(* PLC project Practical Work One, Rexroth ctrlX PLC Engineering ctrlX PLC 1.16.1, author Cedric Lenoir *)
(* stored: creationDateTime 2024-05-03T14:19:29.2185186, version 0.0, modificationDateTime 2024-05-03T14:18:49.029911, organization HEVS *)
(* First Test for Practical Work One *)

TYPE UA_DigitalInput_32 : STRUCT
  Input_0_0 : BOOL;
  Input_0_1 : BOOL;
  Input_0_2 : BOOL;
  Input_0_3 : BOOL;
  Input_0_4 : BOOL;
  Input_0_5 : BOOL;
  Input_0_6 : BOOL;
  Input_0_7 : BOOL;
  Input_1_0 : BOOL;
  Input_1_1 : BOOL;
  Input_1_2 : BOOL;
  Input_1_3 : BOOL;
  Input_1_4 : BOOL;
  Input_1_5 : BOOL;
  Input_1_6 : BOOL;
  Input_1_7 : BOOL;
  Input_2_0 : BOOL;
  Input_2_1 : BOOL;
  Input_2_2 : BOOL;
  Input_2_3 : BOOL;
  Input_2_4 : BOOL;
  Input_2_5 : BOOL;
  Input_2_6 : BOOL;
  Input_2_7 : BOOL;
  Input_3_0 : BOOL;
  Input_3_1 : BOOL;
  Input_3_2 : BOOL;
  Input_3_3 : BOOL;
  Input_3_4 : BOOL;
  Input_3_5 : BOOL;
  Input_3_6 : BOOL;
  Input_3_7 : BOOL;
END_STRUCT;
END_TYPE

TYPE UA_DigitalOutput_32 : STRUCT
  Output_0_0 : BOOL;
  Output_0_1 : BOOL;
  Output_0_2 : BOOL;
  Output_0_3 : BOOL;
  Output_0_4 : BOOL;
  Output_0_5 : BOOL;
  Output_0_6 : BOOL;
  Output_0_7 : BOOL;
  Output_1_0 : BOOL;
  Output_1_1 : BOOL;
  Output_1_2 : BOOL;
  Output_1_3 : BOOL;
  Output_1_4 : BOOL;
  Output_1_5 : BOOL;
  Output_1_6 : BOOL;
  Output_1_7 : BOOL;
  Output_2_0 : BOOL;
  Output_2_1 : BOOL;
  Output_2_2 : BOOL;
  Output_2_3 : BOOL;
  Output_2_4 : BOOL;
  Output_2_5 : BOOL;
  Output_2_6 : BOOL;
  Output_2_7 : BOOL;
  Output_3_0 : BOOL;
  Output_3_1 : BOOL;
  Output_3_2 : BOOL;
  Output_3_3 : BOOL;
  Output_3_4 : BOOL;
  Output_3_5 : BOOL;
  Output_3_6 : BOOL;
  Output_3_7 : BOOL;
END_STRUCT;
END_TYPE

TYPE UA_ButtonAndSignal : STRUCT
  In_Estop : BOOL;
  In_Reset : BOOL;
  In_Start : BOOL;
  In_Stop : BOOL;
  Out_Idle : BOOL;
  Out_Execute : BOOL;
  Out_Stopped : BOOL;
END_STRUCT;
END_TYPE

TYPE UA_O300_DL : STRUCT
  Value : WORD;
  BCD1 : BOOL;
  Q : BOOL;
  A : BOOL;
END_STRUCT;
END_TYPE

TYPE UA_O300_ZL : STRUCT
  BCD1 : BOOL;
  Q : BOOL;
  A : BOOL;
END_STRUCT;
END_TYPE

TYPE UA_U300_D50 : STRUCT
  Value : DWORD;
  Scale : SINT;
  SSC1 : BOOL;
  SSC2 : BOOL;
  Q : BOOL;
  A : BOOL;
  SSC4 : BOOL;
END_STRUCT;
END_TYPE

(* www.hevs.ch Institut Systemes Industriels Project: Projet No: PW Move Absolute Author: Cedric Lenoir Date: 2023 October 16 Summary: List of commands for MoveAbsolute *)
TYPE ST_PlcOpenFbs : STRUCT
  bEnableRemote : BOOL;  (* If TRUE, the FB are driven manually from the HMI *)
  bEnableReadStatus : BOOL;
  bEnableReadPosition : BOOL;
  bEnableReadVelocity : BOOL;
  bMoveAbs : BOOL;
  bStop : BOOL;
  bPowerOn : BOOL;
  bReset : BOOL;
  strGetAxisStatus : STRING;  (* From arAxisStatus_gb[1].Data.PLCopenState; Exist in Data Layer too, s=motion/axs/Axis_X/state/opstate/plcopen *)
END_STRUCT;
END_TYPE

TYPE UA_U300_P50 : STRUCT
  Value : DWORD;
  Scale : SINT;
  SSC1 : BOOL;
  SSC2 : BOOL;
  Q : BOOL;
  A : BOOL;
  SSC4 : BOOL;
END_STRUCT;
END_TYPE

TYPE UA_Schunk_mms : STRUCT
  Value : WORD;
END_STRUCT;
END_TYPE

TYPE UA_Balluf_bcm0002 : STRUCT
  Data_1 : REAL;
  Data_2 : REAL;
  Data_3 : REAL;
  Temperature : REAL;
  Status : DWORD;
END_STRUCT;
END_TYPE

TYPE UA_Festo : STRUCT
  SetOut : BOOL;
END_STRUCT;
END_TYPE

TYPE UA_AnalogIn : STRUCT
  IW_04 : WORD;
  IW_06 : WORD;
  IW_08 : WORD;
  IW_10 : WORD;
  IW_12 : WORD;
  IW_14 : WORD;
  IW_16 : WORD;
  IW_18 : WORD;
END_STRUCT;
END_TYPE

TYPE UA_AnalogOut : STRUCT
  QW_04 : WORD;
  QW_06 : WORD;
  QW_08 : WORD;
  QW_10 : WORD;
END_STRUCT;
END_TYPE

TYPE UA_AboxInterface : STRUCT
  uaButtonAndSignal : UA_ButtonAndSignal;
  uaAnalogIn : UA_AnalogIn;
  uaAnalogOut : UA_AnalogOut;
  uaDigitalIn : UA_DigitalInput_32;
  uaDigitalOut : UA_DigitalOutput_32;
  uaO300_DL_Optic : UA_O300_DL;
  uaO300_ZL_Optic : UA_O300_ZL;
  uaU300_D50_Sound : UA_U300_D50;
  uaU300_P50_Sound : UA_U300_P50;
  uaSchunk : UA_Schunk_mms;
  uaSchunkGripper : UA_Festo;
  uaAccelerometer : UA_Balluf_bcm0002;
END_STRUCT;
END_TYPE

(* www.hevs.ch Institut Systemes Industriels Project: Projet No: PW Move Absolute Author: Cedric Lenoir Date: 2023 October 16 Summary: List of dynamic parameters for Move Absolute *)
TYPE ST_SetMotionParam : STRUCT
  rPosition_mm : LREAL;
  rVeloctiy_mm_s : LREAL;
  rAcceleration_mm_s2 : LREAL;
  rDeceleration_mm_s2 : LREAL;
  rJerk_mm_s3 : LREAL;
END_STRUCT;
END_TYPE

(* www.hevs.ch Institut Systemes Industriels Project: Projet No: PW Move Absolute Author: Cedric Lenoir Date: 2023 October 16 Summary: State Machine Info *)
TYPE ST_StateMachineInfo : STRUCT
  diState : DINT;
  eState : E_Execute;
  strState : STRING;
END_STRUCT;
END_TYPE

{attribute 'qualified_only'}
{attribute 'strict'}
TYPE E_PackStates : (NotActive := 999, Aborted := 10, Clearing := 20, Stopped := 30, Resetting := 40, Idle := 50, Starting := 60, Stopping := 70, Aborting := 80, Execute := 90, Holding := 100, Held := 110, Unholding := 120, Suspending := 200, Suspended := 210, Unsuspending := 220, Completing := 300, Complete := 310) DINT;
END_TYPE

TYPE ST_PackState : STRUCT
  Aborted : BOOL;
  Clearing : BOOL;
  Stopped : BOOL;
  Resetting : BOOL;
  Idle : BOOL;
  Starting : BOOL;
  Stopping : BOOL;
  Aborting : BOOL;
  Execute : BOOL;
  Holding : BOOL;  (* Held Loop *)
  Held : BOOL;
  Unholding : BOOL;
  Suspending : BOOL;  (* Suspended Loop *)
  Suspended : BOOL;
  Unsuspending : BOOL;
  Completing : BOOL;  (* Complete Loop *)
  Complete : BOOL;
END_STRUCT;
END_TYPE

{attribute 'qualified_only'}
{attribute 'strict'}
TYPE E_Clearing : (Idle := 99);
END_TYPE

{attribute 'qualified_only'}
{attribute 'strict'}
TYPE E_Stopping : (Idle := 99);
END_TYPE

{attribute 'qualified_only'}
{attribute 'strict'}
TYPE E_Aborting : (Idle := 99, Disabled := 1, ErrorStop := 2);
END_TYPE

{attribute 'qualified_only'}
{attribute 'strict'}
TYPE E_Resetting : (Idle := 99, eMotionInit := 10, eMotionInitDone := 20);
END_TYPE

{attribute 'qualified_only'}
{attribute 'strict'}
TYPE E_Starting : (Idle := 99, eMotionStarting := 10, eMotionStartingDone := 20, eMotionStartSetPointBack := 22, eMotionStartSetPointBackDone := 23, eMotionSetSynch := 30, eMotionSetSynchDone := 40);
END_TYPE

TYPE ST_RemoteCyclicSetPosition : STRUCT
  in : ST_RemoteCyclicSetPositionIn;  (* Commands for program *)
  out : ST_RemoteCyclicSetPositionOut;  (* Status for program *)
END_STRUCT;
END_TYPE

TYPE ST_RemoteCyclicSetPositionIn : STRUCT
  lrStartPosition_mm : LREAL;  (* Set init position / Start of profile position *)
  lrEndPosition_mm : LREAL;  (* Set end position / End of profile position *)
  udiCycleTimeMultiplier : UDINT := 1000;  (* Cycle Time Multiplier, default is 1000 for 1000 ms *)
  bActivateCoupling : BOOL;  (* Activate coupling, when TRUE, axis position is set by fbGenerateProfile with 5th order polynomial *)
  bStartForward : BOOL;  (* Start polynomial profile forward *)
  bStartBackward : BOOL;  (* Start polynomial profile backward *)
  lrProfileSetPosition : LREAL;  (* Set Position from Profile generator *)
END_STRUCT;
END_TYPE

TYPE ST_RemoteCyclicSetPositionOut : STRUCT
  bInitDone : BOOL;  (* Init done, ready for cyclic motion *)
  bError : BOOL;  (* There is an error *)
  bFwdDone : BOOL;  (* End of cyclic profile Forward *)
  bBackDone : BOOL;  (* End of cyclic profile Back *)
END_STRUCT;
END_TYPE

{attribute 'qualified_only'}
{attribute 'strict'}
TYPE E_Aborted : (Idle := 99, Disabled := 1, ErrorStop := 2);
END_TYPE

(* www.hevs.ch Institut Systemes Industriels Project: Projet No: PW Move Absolute Author: Cedric Lenoir Date: 2024 April 02 Summary: Template of a program using PLCopen on partial Pack State Use a Cyclic Setpoint for motion in Pack Execute. *)
PROGRAM PRG_CyclicSetPoint
  VAR
    uliCount : ULINT;
    bInitDone : BOOL;
    fbPackStates : FB_PackStates;  (* Pack Partial state machine *)
    eAborting : E_Aborting;
    eAborted : E_Aborted;
    eClearing : E_Clearing;
    eResetting : E_Resetting;
    eStarting : E_Starting;
    eStopping : E_Stopping;
    stPlcOpenFbs : ST_PlcOpenFbs;  (* List of Structures *)
    stSetMotionParam : ST_SetMotionParam := (rVeloctiy_mm_s := 2000, rAcceleration_mm_s2 := 1000, rDeceleration_mm_s2 := 1000, rJerk_mm_s3 := 1);
    stStateMachineInfo : ST_StateMachineInfo;
    mcReadActualPosition : MC_ReadActualPosition;  (* List of Function Blocks *)
    mcReadActualVelocity : MC_ReadActualVelocity;
    mcReadStatus : MC_ReadStatus;
    mcPower : MC_Power;
    mcMoveAbsolute : MC_MoveAbsolute;
    mcStop : MC_Stop := (Deceleration := 1);
    mcReset : MC_Reset;
    mcCyclicSetPoint : MB_CyclicSetPoint;
    fbGenerateProfile : FB_GenerateProfile;  (* Set point generator *)
  END_VAR

                    (*
    Some inits independant of the Main State Machine
*)
IF NOT bInitDone THEN
	bInitDone := TRUE;
    stPlcOpenFbs.bEnableReadStatus := TRUE;
    stPlcOpenFbs.bEnableReadPosition := TRUE;
    stPlcOpenFbs.bEnableReadVelocity := TRUE;
END_IF

(*
    Remote conditions
*)
IF stPlcOpenFbs.bEnableRemote THEN
    IF mcMoveAbsolute.Done THEN
        stPlcOpenFbs.bMoveAbs := FALSE;
    END_IF
    IF mcStop.Done THEN
        stPlcOpenFbs.bStop := FALSE;
        stPlcOpenFbs.bMoveAbs := FALSE;
    END_IF
END_IF

// If remote, pack states are disabled
fbPackStates.SoftEstop := mcReadStatus.ErrorStop;
fbPackStates(Enable := NOT stPlcOpenFbs.bEnableRemote,
			 remote := GVL_Abox.uaAboxInterface.uaButtonAndSignal);
			 
(*
	Basically, only Acting state are used, wait state are doing nothing
*)

IF fbPackStates.state.Aborting THEN
	IF mcReadStatus.ErrorStop THEN
		fbPackStates.Aborting_SC := FALSE;
	ELSE
		fbPackStates.Aborting_SC := TRUE;
	END_IF
ELSE
	;
END_IF

IF fbPackStates.state.Aborted THEN
	CASE eAborted OF
		E_Aborted.Idle :
			IF mcReadStatus.Disabled THEN
				eAborted := E_Aborted.Disabled;
			ELSIF mcReadStatus.ErrorStop THEN
				eAborted := E_Aborted.ErrorStop;
			END_IF
		E_Aborted.Disabled :
			IF mcReadStatus.ErrorStop THEN
				eAborted := E_Aborted.ErrorStop;
			END_IF
		E_Aborted.ErrorStop :
			IF mcReadStatus.Disabled THEN
				eAborted := E_Aborted.Disabled;
			END_IF
	END_CASE
ELSE
	eAborted := E_Aborted.Idle;
END_IF

IF fbPackStates.state.Clearing THEN
	IF mcReadStatus.Standstill THEN
		fbPackStates.Clearing_SC := TRUE;
	ELSE
		fbPackStates.Clearing_SC := FALSE;
	END_IF
ELSE
	;
END_IF

IF fbPackStates.state.Stopping THEN
	IF mcReadStatus.Standstill THEN
		fbPackStates.Stopping_SC := TRUE;
	ELSE
		fbPackStates.Stopping_SC := FALSE;
	END_IF
ELSE
	;
END_IF

IF fbPackStates.state.Resetting THEN
	fbPackStates.Resetting_SC := FALSE;
	CASE eResetting OF
		E_Resetting.Idle :
            stSetMotionParam.rPosition_mm := 50;
			stSetMotionParam.rVeloctiy_mm_s := 2000;  
			eResetting := E_Resetting.eMotionInit;

		E_Resetting.eMotionInit :
			IF mcMoveAbsolute.Done THEN
				eResetting := E_Resetting.eMotionInitDone; 
			END_IF

		E_Resetting.eMotionInitDone :
			;;
	END_CASE
	 
	IF eResetting = E_Resetting.eMotionInitDone THEN
		fbPackStates.Resetting_SC := TRUE;
	END_IF
ELSE
	eResetting := E_Resetting.Idle;
END_IF

IF fbPackStates.state.Starting THEN
	fbPackStates.Starting_SC := FALSE;
	CASE eStarting OF
		E_Starting.Idle :
            stSetMotionParam.rPosition_mm := GVL_CyclSetPoint.stRemote.in.lrStartPosition_mm;
			stSetMotionParam.rVeloctiy_mm_s := 2000;  
			eStarting := E_Starting.eMotionStarting;

		E_Starting.eMotionStarting :
			IF mcMoveAbsolute.Done THEN
				eStarting := E_Starting.eMotionStartingDone; 
			END_IF

		E_Starting.eMotionStartingDone :
			IF mcReadStatus.Standstill THEN
				eStarting := E_Starting.eMotionStartSetPointBack;
			END_IF
			
		E_Starting.eMotionStartSetPointBack :
			IF GVL_CyclSetPoint.stRemote.out.bBackDone THEN
				eStarting := E_Starting.eMotionStartSetPointBackDone;
			END_IF
	
		E_Starting.eMotionStartSetPointBackDone :
			eStarting := E_Starting.eMotionSetSynch;

		E_Starting.eMotionSetSynch :
			IF mcReadStatus.DiscreteMotion THEN
				eStarting := E_Starting.eMotionSetSynchDone;
			END_IF
			
		E_Starting.eMotionSetSynchDone :
			;			
			
	END_CASE
	 
	IF eStarting = E_Starting.eMotionSetSynchDone THEN
		fbPackStates.Starting_SC := TRUE;
	END_IF
ELSE
	eStarting := E_Starting.Idle;
END_IF

IF fbPackStates.state.Execute THEN
	fbPackStates.Execute_SC := FALSE;
	(*
		Execute State Machine.
	*)
	CASE stStateMachineInfo.eState OF
		E_Execute.eIdle :
			stStateMachineInfo.strState := 'Idle';
			IF mcCyclicSetPoint.InOperation THEN
				// Set as default value in GVL_CyclSetPoint
				// GVL_CyclSetPoint.stRemote.in.lrEndPosition_mm := 100; 
				stStateMachineInfo.eState := E_Execute.eMotionFwd;
			END_IF

		E_Execute.eMotionFwd :
			stStateMachineInfo.strState := 'Motion One';
			IF GVL_CyclSetPoint.stRemote.out.bFwdDone THEN
				stStateMachineInfo.eState := E_Execute.eMotionFwdDone; 
			END_IF

		E_Execute.eMotionFwdDone :
			stStateMachineInfo.strState := 'Motion One Done';
			IF mcCyclicSetPoint.InOperation THEN
				// Set as default value in GVL_CyclSetPoint
				// GVL_CyclSetPoint.stRemote.in.lrStartPosition_mm := 50;
				stStateMachineInfo.eState := E_Execute.eMotionBack;
			END_IF

		E_Execute.eMotionBack :
			stStateMachineInfo.strState := 'Motion Two';
			IF GVL_CyclSetPoint.stRemote.out.bBackDone THEN
				stStateMachineInfo.eState := E_Execute.eMotionBackDone; 
			END_IF

		E_Execute.eMotionBackDone :
			stStateMachineInfo.strState := 'Motion Two Done'; 
			stStateMachineInfo.eState :=E_Execute.eIdle; 

	END_CASE
	;
ELSE
	stStateMachineInfo.eState := E_Execute.eIdle;
END_IF

IF fbPackStates.state.Holding THEN
	fbPackStates.Holding_SC := TRUE;
ELSE
	;
END_IF

IF fbPackStates.state.Unholding THEN
	fbPackStates.Unholding_SC := TRUE;
ELSE
	;
END_IF

(*
    Get state machine in a DINT format
*)
stStateMachineInfo.diState := stStateMachineInfo.eState;

(*
    Call all Function Blocks at the end of the program
    This is a good practice.
*)
mcReadStatus(Axis := GVL_AxisDefines.X_Axis,
             Enable := stPlcOpenFbs.bEnableReadStatus);

mcReadActualPosition(Axis := GVL_AxisDefines.X_Axis,
                     Enable := stPlcOpenFbs.bEnableReadPosition);
                                         
mcReadActualVelocity(Axis := GVL_AxisDefines.X_Axis,
                     Enable := stPlcOpenFbs.bEnableReadVelocity);

mcPower(Axis := GVL_AxisDefines.X_Axis,
        Enable := (stPlcOpenFbs.bPowerOn AND stPlcOpenFbs.bEnableRemote) OR
                   		NOT stPlcOpenFbs.bEnableRemote AND 
				   		NOT (fbPackStates.state.Aborting OR
                             fbPackStates.state.Aborted));

mcMoveAbsolute(Axis := GVL_AxisDefines.X_Axis,
               Position := stSetMotionParam.rPosition_mm,
               Velocity := stSetMotionParam.rVeloctiy_mm_s,
               Acceleration := stSetMotionParam.rAcceleration_mm_s2,
               Deceleration := stSetMotionParam.rDeceleration_mm_s2,
               Jerk := stSetMotionParam.rJerk_mm_s3,
               Execute := (stPlcOpenFbs.bMoveAbs AND stPlcOpenFbs.bEnableRemote)    OR
                          (eResetting = E_Resetting.eMotionInit)                    OR
						  (eStarting = E_Starting.eMotionStarting));               

// Note that a stop without deceleration leads to an error!!
mcStop(Axis := GVL_AxisDefines.X_Axis,
       Execute := (stPlcOpenFbs.bStop AND stPlcOpenFbs.bEnableRemote) OR
                   fbPackStates.state.Stopping);

mcReset(Axis := GVL_AxisDefines.X_Axis,
        Execute := (stPlcOpenFbs.bReset AND stPlcOpenFbs.bEnableRemote) OR
                    fbPackStates.state.Aborting                         OR
                    eAborted = E_Aborted.ErrorStop);
					
(*
	Set Point Generator
*)
mcCyclicSetPoint.Execute := (stPlcOpenFbs.bEnableRemote AND GVL_CyclSetPoint.stRemote.in.bActivateCoupling) OR
                            (eStarting = E_Starting.eMotionSetSynch);
mcCyclicSetPoint.SetPoint := GVL_CyclSetPoint.stRemote.in.lrProfileSetPosition;
mcCyclicSetPoint(Axis := GVL_AxisDefines.X_Axis);

fbGenerateProfile(bStartForward := (stPlcOpenFbs.bEnableRemote AND GVL_CyclSetPoint.stRemote.in.bStartForward) OR
                                   (stStateMachineInfo.eState = E_Execute.eMotionFwd),
                  bStartBackward := (stPlcOpenFbs.bEnableRemote AND GVL_CyclSetPoint.stRemote.in.bStartBackward) OR
                                    (eStarting = E_Starting.eMotionStartSetPointBack) OR
                                    (stStateMachineInfo.eState = E_Execute.eMotionBack),
                  startPosition_mm := GVL_CyclSetPoint.stRemote.in.lrStartPosition_mm,
                  endPosition_mm := GVL_CyclSetPoint.stRemote.in.lrEndPosition_mm,
                  udiCyclTime_ms := GVL_CyclSetPoint.MOTION_CYCLE_TIME_ms,
                  udiCycleTimeMult := GVL_CyclSetPoint.stRemote.in.udiCycleTimeMultiplier, // Could be a parameter latter when all is working
                  arGoToPos := GVL_CyclSetPoint.arGoToPosition,
                  arReturnFromPos := GVL_CyclSetPoint.arReturnFromPosition,
                  lrSetPosition => GVL_CyclSetPoint.stRemote.in.lrProfileSetPosition,
                  bDoneForward => GVL_CyclSetPoint.stRemote.out.bFwdDone,
                  bDoneBackward => GVL_CyclSetPoint.stRemote.out.bBackDone);					
					
                   
                  
END_PROGRAM

PROGRAM PRG_MapBox
  VAR
    UA_ReadCounterFromStation : DINT;  (* Write from Siemens to ctrX Core Used to check if read is running *)
    UA_ButtonAndSignal_In_Estop : BOOL;
    UA_ButtonAndSignal_In_Reset : BOOL;
    UA_ButtonAndSignal_In_Start : BOOL;
    UA_ButtonAndSignal_In_Stop : BOOL;
    UA_Balluf_bcm0002_Data_1 : REAL;
    UA_Balluf_bcm0002_Data_2 : REAL;
    UA_Balluf_bcm0002_Data_3 : REAL;
    UA_Balluf_bcm0002_Temperature : REAL;
    UA_Balluf_bcm0002_Status : DWORD;
    UA_Festo_SetOut : BOOL;
    UA_O300_DL_Value : WORD;
    UA_O300_DL_BCD1 : BOOL;
    UA_O300_DL_Q : BOOL;
    UA_O300_DL_A : BOOL;
    UA_O300_ZL_BCD1 : BOOL;
    UA_O300_ZL_Q : BOOL;
    UA_O300_ZL_A : BOOL;
    UA_U300_D50_Value : DWORD;
    UA_U300_D50_Scale : SINT;
    UA_U300_D50_SSC1 : BOOL;
    UA_U300_D50_SSC2 : BOOL;
    UA_U300_D50_Q : BOOL;
    UA_U300_D50_A : BOOL;
    UA_U300_D50_SSC4 : BOOL;
    UA_U300_P50_Value : DWORD;
    UA_U300_P50_Scale : SINT;
    UA_U300_P50_SSC1 : BOOL;
    UA_U300_P50_SSC2 : BOOL;
    UA_U300_P50_Q : BOOL;
    UA_U300_P50_A : BOOL;
    UA_U300_P50_SSC4 : BOOL;
    UA_DigitalInput_32_Input_0_0 : BOOL;
    UA_DigitalInput_32_Input_0_1 : BOOL;
    UA_DigitalInput_32_Input_0_2 : BOOL;
    UA_DigitalInput_32_Input_0_3 : BOOL;
    UA_DigitalInput_32_Input_0_4 : BOOL;
    UA_DigitalInput_32_Input_0_5 : BOOL;
    UA_DigitalInput_32_Input_0_6 : BOOL;
    UA_DigitalInput_32_Input_0_7 : BOOL;
    UA_DigitalInput_32_Input_1_0 : BOOL;
    UA_DigitalInput_32_Input_1_1 : BOOL;
    UA_DigitalInput_32_Input_1_2 : BOOL;
    UA_DigitalInput_32_Input_1_3 : BOOL;
    UA_DigitalInput_32_Input_1_4 : BOOL;
    UA_DigitalInput_32_Input_1_5 : BOOL;
    UA_DigitalInput_32_Input_1_6 : BOOL;
    UA_DigitalInput_32_Input_1_7 : BOOL;
    UA_DigitalInput_32_Input_2_0 : BOOL;
    UA_DigitalInput_32_Input_2_1 : BOOL;
    UA_DigitalInput_32_Input_2_2 : BOOL;
    UA_DigitalInput_32_Input_2_3 : BOOL;
    UA_DigitalInput_32_Input_2_4 : BOOL;
    UA_DigitalInput_32_Input_2_5 : BOOL;
    UA_DigitalInput_32_Input_2_6 : BOOL;
    UA_DigitalInput_32_Input_2_7 : BOOL;
    UA_DigitalInput_32_Input_3_0 : BOOL;
    UA_DigitalInput_32_Input_3_1 : BOOL;
    UA_DigitalInput_32_Input_3_2 : BOOL;
    UA_DigitalInput_32_Input_3_3 : BOOL;
    UA_DigitalInput_32_Input_3_4 : BOOL;
    UA_DigitalInput_32_Input_3_5 : BOOL;
    UA_DigitalInput_32_Input_3_6 : BOOL;
    UA_DigitalInput_32_Input_3_7 : BOOL;
    UA_WriteCounterToStation : DINT;  (* Siemens Read from ctrX Core Used to check if write is running *)
    UA_ButtonAndSignal_Out_Idle : BOOL;
    UA_ButtonAndSignal_Out_Execute : BOOL;
    UA_ButtonAndSignal_Out_Stopped : BOOL;
    UA_Schunk_mms_Value : WORD;
    UA_DigitalOutput_32_Output_0_0 : BOOL;
    UA_DigitalOutput_32_Output_0_1 : BOOL;
    UA_DigitalOutput_32_Output_0_2 : BOOL;
    UA_DigitalOutput_32_Output_0_3 : BOOL;
    UA_DigitalOutput_32_Output_0_4 : BOOL;
    UA_DigitalOutput_32_Output_0_5 : BOOL;
    UA_DigitalOutput_32_Output_0_6 : BOOL;
    UA_DigitalOutput_32_Output_0_7 : BOOL;
    UA_DigitalOutput_32_Output_1_0 : BOOL;
    UA_DigitalOutput_32_Output_1_1 : BOOL;
    UA_DigitalOutput_32_Output_1_2 : BOOL;
    UA_DigitalOutput_32_Output_1_3 : BOOL;
    UA_DigitalOutput_32_Output_1_4 : BOOL;
    UA_DigitalOutput_32_Output_1_5 : BOOL;
    UA_DigitalOutput_32_Output_1_6 : BOOL;
    UA_DigitalOutput_32_Output_1_7 : BOOL;
    UA_DigitalOutput_32_Output_2_0 : BOOL;
    UA_DigitalOutput_32_Output_2_1 : BOOL;
    UA_DigitalOutput_32_Output_2_2 : BOOL;
    UA_DigitalOutput_32_Output_2_3 : BOOL;
    UA_DigitalOutput_32_Output_2_4 : BOOL;
    UA_DigitalOutput_32_Output_2_5 : BOOL;
    UA_DigitalOutput_32_Output_2_6 : BOOL;
    UA_DigitalOutput_32_Output_2_7 : BOOL;
    UA_DigitalOutput_32_Output_3_0 : BOOL;
    UA_DigitalOutput_32_Output_3_1 : BOOL;
    UA_DigitalOutput_32_Output_3_2 : BOOL;
    UA_DigitalOutput_32_Output_3_3 : BOOL;
    UA_DigitalOutput_32_Output_3_4 : BOOL;
    UA_DigitalOutput_32_Output_3_5 : BOOL;
    UA_DigitalOutput_32_Output_3_6 : BOOL;
    UA_DigitalOutput_32_Output_3_7 : BOOL;
  END_VAR

                        (*
        Values from Profinet Station
    *)
    
    // Get Value from Profinet Station with UA Client Write
	GVL_Abox.uaAboxInterface.uaButtonAndSignal.In_Estop     := UA_ButtonAndSignal_In_Estop;
	GVL_Abox.uaAboxInterface.uaButtonAndSignal.In_Reset     := UA_ButtonAndSignal_In_Reset;
	GVL_Abox.uaAboxInterface.uaButtonAndSignal.In_Start     := UA_ButtonAndSignal_In_Start;
	GVL_Abox.uaAboxInterface.uaButtonAndSignal.In_Stop      := UA_ButtonAndSignal_In_Stop;
    // Values from Balluff accelerometer
    GVL_Abox.uaAboxInterface.uaAccelerometer.Data_1         := UA_Balluf_bcm0002_Data_1;
    GVL_Abox.uaAboxInterface.uaAccelerometer.Data_2         := UA_Balluf_bcm0002_Data_1;
    GVL_Abox.uaAboxInterface.uaAccelerometer.Data_3         := UA_Balluf_bcm0002_Data_1;
    GVL_Abox.uaAboxInterface.uaAccelerometer.Status         := UA_Balluf_bcm0002_Status;
    GVL_Abox.uaAboxInterface.uaAccelerometer.Temperature    := UA_Balluf_bcm0002_Temperature;

    // Values from Baumer O300 DL
    GVL_Abox.uaAboxInterface.uaO300_DL_Optic.Value          := UA_O300_DL_Value;                
    GVL_Abox.uaAboxInterface.uaO300_DL_Optic.A              := UA_O300_DL_A;                
    GVL_Abox.uaAboxInterface.uaO300_DL_Optic.Q              := UA_O300_DL_Q;                
    GVL_Abox.uaAboxInterface.uaO300_DL_Optic.BCD1           := UA_O300_DL_BCD1;                

    // Values from Baumer O300 ZL                
    GVL_Abox.uaAboxInterface.uaO300_ZL_Optic.A              := UA_O300_ZL_A;                
    GVL_Abox.uaAboxInterface.uaO300_ZL_Optic.Q              := UA_O300_ZL_Q;                
    GVL_Abox.uaAboxInterface.uaO300_ZL_Optic.BCD1           := UA_O300_ZL_BCD1;                

    // Values from Baumer U300 D50
    GVL_Abox.uaAboxInterface.uaU300_D50_Sound.Value         := UA_U300_D50_Value;  
    GVL_Abox.uaAboxInterface.uaU300_D50_Sound.A             := UA_U300_D50_A;  
    GVL_Abox.uaAboxInterface.uaU300_D50_Sound.Q             := UA_U300_D50_Q;  
    GVL_Abox.uaAboxInterface.uaU300_D50_Sound.Scale         := UA_U300_D50_Scale;  
    GVL_Abox.uaAboxInterface.uaU300_D50_Sound.SSC1          := UA_U300_D50_SSC1;  
    GVL_Abox.uaAboxInterface.uaU300_D50_Sound.SSC2          := UA_U300_D50_SSC2;  
    GVL_Abox.uaAboxInterface.uaU300_D50_Sound.SSC4          := UA_U300_D50_SSC4;  
    
    // Values from Baumer U300 P50
    GVL_Abox.uaAboxInterface.uaU300_P50_Sound.Value         := UA_U300_P50_Value;  
    GVL_Abox.uaAboxInterface.uaU300_P50_Sound.A             := UA_U300_P50_A;  
    GVL_Abox.uaAboxInterface.uaU300_P50_Sound.Q             := UA_U300_P50_Q;  
    GVL_Abox.uaAboxInterface.uaU300_P50_Sound.Scale         := UA_U300_P50_Scale;  
    GVL_Abox.uaAboxInterface.uaU300_P50_Sound.SSC1          := UA_U300_P50_SSC1;  
    GVL_Abox.uaAboxInterface.uaU300_P50_Sound.SSC2          := UA_U300_P50_SSC2;  
    GVL_Abox.uaAboxInterface.uaU300_P50_Sound.SSC4          := UA_U300_P50_SSC4;  
    
    // Values from Gripper sensor
    GVL_Abox.uaAboxInterface.uaSchunk.Value                 := UA_Schunk_mms_Value;  
    
    // Get 32 Digital Input
    GVL_Abox.uaAboxInterface.uaDigitalIn.Input_0_0          := UA_DigitalInput_32_Input_0_0;
    GVL_Abox.uaAboxInterface.uaDigitalIn.Input_0_1          := UA_DigitalInput_32_Input_0_1;
    GVL_Abox.uaAboxInterface.uaDigitalIn.Input_0_2          := UA_DigitalInput_32_Input_0_2;
    GVL_Abox.uaAboxInterface.uaDigitalIn.Input_0_3          := UA_DigitalInput_32_Input_0_3;
    GVL_Abox.uaAboxInterface.uaDigitalIn.Input_0_4          := UA_DigitalInput_32_Input_0_4;
    GVL_Abox.uaAboxInterface.uaDigitalIn.Input_0_5          := UA_DigitalInput_32_Input_0_5;
    GVL_Abox.uaAboxInterface.uaDigitalIn.Input_0_6          := UA_DigitalInput_32_Input_0_6;
    GVL_Abox.uaAboxInterface.uaDigitalIn.Input_0_7          := UA_DigitalInput_32_Input_0_7;
    GVL_Abox.uaAboxInterface.uaDigitalIn.Input_1_0          := UA_DigitalInput_32_Input_1_0;
    GVL_Abox.uaAboxInterface.uaDigitalIn.Input_1_1          := UA_DigitalInput_32_Input_1_1;
    GVL_Abox.uaAboxInterface.uaDigitalIn.Input_1_2          := UA_DigitalInput_32_Input_1_2;
    GVL_Abox.uaAboxInterface.uaDigitalIn.Input_1_3          := UA_DigitalInput_32_Input_1_3;
    GVL_Abox.uaAboxInterface.uaDigitalIn.Input_1_4          := UA_DigitalInput_32_Input_1_4;
    GVL_Abox.uaAboxInterface.uaDigitalIn.Input_1_5          := UA_DigitalInput_32_Input_1_5;
    GVL_Abox.uaAboxInterface.uaDigitalIn.Input_1_6          := UA_DigitalInput_32_Input_1_6;
    GVL_Abox.uaAboxInterface.uaDigitalIn.Input_1_7          := UA_DigitalInput_32_Input_1_7;
    GVL_Abox.uaAboxInterface.uaDigitalIn.Input_2_0          := UA_DigitalInput_32_Input_2_0;
    GVL_Abox.uaAboxInterface.uaDigitalIn.Input_2_1          := UA_DigitalInput_32_Input_2_1;
    GVL_Abox.uaAboxInterface.uaDigitalIn.Input_2_2          := UA_DigitalInput_32_Input_2_2;
    GVL_Abox.uaAboxInterface.uaDigitalIn.Input_2_3          := UA_DigitalInput_32_Input_2_3;
    GVL_Abox.uaAboxInterface.uaDigitalIn.Input_2_4          := UA_DigitalInput_32_Input_2_4;
    GVL_Abox.uaAboxInterface.uaDigitalIn.Input_2_5          := UA_DigitalInput_32_Input_2_5;
    GVL_Abox.uaAboxInterface.uaDigitalIn.Input_2_6          := UA_DigitalInput_32_Input_2_6;
    GVL_Abox.uaAboxInterface.uaDigitalIn.Input_2_7          := UA_DigitalInput_32_Input_2_7;
    GVL_Abox.uaAboxInterface.uaDigitalIn.Input_3_0          := UA_DigitalInput_32_Input_3_0;
    GVL_Abox.uaAboxInterface.uaDigitalIn.Input_3_1          := UA_DigitalInput_32_Input_3_1;
    GVL_Abox.uaAboxInterface.uaDigitalIn.Input_3_2          := UA_DigitalInput_32_Input_3_2;
    GVL_Abox.uaAboxInterface.uaDigitalIn.Input_3_3          := UA_DigitalInput_32_Input_3_3;
    GVL_Abox.uaAboxInterface.uaDigitalIn.Input_3_4          := UA_DigitalInput_32_Input_3_4;
    GVL_Abox.uaAboxInterface.uaDigitalIn.Input_3_5          := UA_DigitalInput_32_Input_3_5;
    GVL_Abox.uaAboxInterface.uaDigitalIn.Input_3_6          := UA_DigitalInput_32_Input_3_6;
    GVL_Abox.uaAboxInterface.uaDigitalIn.Input_3_7          := UA_DigitalInput_32_Input_3_7;
    
    (*
        Values to Profinet Station
    *)
	UA_WriteCounterToStation := UA_WriteCounterToStation + 1;

    // Set Visual Signals
	UA_ButtonAndSignal_Out_Execute 	:= GVL_Abox.uaAboxInterface.uaButtonAndSignal.Out_Execute;
	UA_ButtonAndSignal_Out_Idle 	:= GVL_Abox.uaAboxInterface.uaButtonAndSignal.Out_Idle;
	UA_ButtonAndSignal_Out_Stopped	:= GVL_Abox.uaAboxInterface.uaButtonAndSignal.Out_Stopped;
    
    // Set Gripper value
    UA_Festo_SetOut                 := GVL_Abox.uaAboxInterface.uaSchunkGripper.SetOut;
    
    // Set 32 digital outputs
    UA_DigitalOutput_32_Output_0_0  := GVL_Abox.uaAboxInterface.uaDigitalOut.Output_0_0;
    UA_DigitalOutput_32_Output_0_1  := GVL_Abox.uaAboxInterface.uaDigitalOut.Output_0_1;
    UA_DigitalOutput_32_Output_0_2  := GVL_Abox.uaAboxInterface.uaDigitalOut.Output_0_2;
    UA_DigitalOutput_32_Output_0_3  := GVL_Abox.uaAboxInterface.uaDigitalOut.Output_0_3;
    UA_DigitalOutput_32_Output_0_4  := GVL_Abox.uaAboxInterface.uaDigitalOut.Output_0_4;
    UA_DigitalOutput_32_Output_0_5  := GVL_Abox.uaAboxInterface.uaDigitalOut.Output_0_5;
    UA_DigitalOutput_32_Output_0_6  := GVL_Abox.uaAboxInterface.uaDigitalOut.Output_0_6;
    UA_DigitalOutput_32_Output_0_7  := GVL_Abox.uaAboxInterface.uaDigitalOut.Output_0_7;
    UA_DigitalOutput_32_Output_1_0  := GVL_Abox.uaAboxInterface.uaDigitalOut.Output_1_0;
    UA_DigitalOutput_32_Output_1_1  := GVL_Abox.uaAboxInterface.uaDigitalOut.Output_1_1;
    UA_DigitalOutput_32_Output_1_2  := GVL_Abox.uaAboxInterface.uaDigitalOut.Output_1_2;
    UA_DigitalOutput_32_Output_1_3  := GVL_Abox.uaAboxInterface.uaDigitalOut.Output_1_3;
    UA_DigitalOutput_32_Output_1_4  := GVL_Abox.uaAboxInterface.uaDigitalOut.Output_1_4;
    UA_DigitalOutput_32_Output_1_5  := GVL_Abox.uaAboxInterface.uaDigitalOut.Output_1_5;
    UA_DigitalOutput_32_Output_1_6  := GVL_Abox.uaAboxInterface.uaDigitalOut.Output_1_6;
    UA_DigitalOutput_32_Output_1_7  := GVL_Abox.uaAboxInterface.uaDigitalOut.Output_1_7;
    UA_DigitalOutput_32_Output_2_0  := GVL_Abox.uaAboxInterface.uaDigitalOut.Output_2_0;
    UA_DigitalOutput_32_Output_2_1  := GVL_Abox.uaAboxInterface.uaDigitalOut.Output_2_1;
    UA_DigitalOutput_32_Output_2_2  := GVL_Abox.uaAboxInterface.uaDigitalOut.Output_2_2;
    UA_DigitalOutput_32_Output_2_3  := GVL_Abox.uaAboxInterface.uaDigitalOut.Output_2_3;
    UA_DigitalOutput_32_Output_2_4  := GVL_Abox.uaAboxInterface.uaDigitalOut.Output_2_4;
    UA_DigitalOutput_32_Output_2_5  := GVL_Abox.uaAboxInterface.uaDigitalOut.Output_2_5;
    UA_DigitalOutput_32_Output_2_6  := GVL_Abox.uaAboxInterface.uaDigitalOut.Output_2_6;
    UA_DigitalOutput_32_Output_2_7  := GVL_Abox.uaAboxInterface.uaDigitalOut.Output_2_7;
    UA_DigitalOutput_32_Output_3_0  := GVL_Abox.uaAboxInterface.uaDigitalOut.Output_3_0;
    UA_DigitalOutput_32_Output_3_1  := GVL_Abox.uaAboxInterface.uaDigitalOut.Output_3_1;
    UA_DigitalOutput_32_Output_3_2  := GVL_Abox.uaAboxInterface.uaDigitalOut.Output_3_2;
    UA_DigitalOutput_32_Output_3_3  := GVL_Abox.uaAboxInterface.uaDigitalOut.Output_3_3;
    UA_DigitalOutput_32_Output_3_4  := GVL_Abox.uaAboxInterface.uaDigitalOut.Output_3_4;
    UA_DigitalOutput_32_Output_3_5  := GVL_Abox.uaAboxInterface.uaDigitalOut.Output_3_5;
    UA_DigitalOutput_32_Output_3_6  := GVL_Abox.uaAboxInterface.uaDigitalOut.Output_3_6;
    UA_DigitalOutput_32_Output_3_7  := GVL_Abox.uaAboxInterface.uaDigitalOut.Output_3_7;
    
PRG_CHECK_IO();
                  
END_PROGRAM

PROGRAM PRG_CHECK_IO
  VAR
    testButton_1 : BOOL;
    testButton_2 : BOOL;
    testButton_3 : BOOL;
    clignote : TON;
    changeMeSlow : BOOL;
    clignoteSlow : TON;
    changeMe : BOOL;
    NotResetTest : BOOL := TRUE;
  END_VAR

                    testButton_1 := GVL_Abox.uaAboxInterface.uaButtonAndSignal.In_Reset;
testButton_2 := GVL_Abox.uaAboxInterface.uaButtonAndSignal.In_Start;
testButton_3 := GVL_Abox.uaAboxInterface.uaButtonAndSignal.In_Stop;

IF GVL_Abox.uaAboxInterface.uaButtonAndSignal.In_Reset AND
   NotResetTest										   THEN
	NotResetTest := FALSE;
	
    GVL_Abox.uaAboxInterface.uaSchunkGripper.SetOut := FALSE;
    
    GVL_Abox.uaAboxInterface.uaButtonAndSignal.Out_Execute := FALSE;	
    GVL_Abox.uaAboxInterface.uaButtonAndSignal.Out_Idle := FALSE;	
    GVL_Abox.uaAboxInterface.uaButtonAndSignal.Out_Stopped := FALSE;	

    GVL_Abox.uaAboxInterface.uaDigitalOut.Output_0_0 := FALSE;
    GVL_Abox.uaAboxInterface.uaDigitalOut.Output_0_1 := FALSE;
    GVL_Abox.uaAboxInterface.uaDigitalOut.Output_0_2 := FALSE;
    GVL_Abox.uaAboxInterface.uaDigitalOut.Output_0_3 := FALSE;
    GVL_Abox.uaAboxInterface.uaDigitalOut.Output_0_4 := FALSE;
    GVL_Abox.uaAboxInterface.uaDigitalOut.Output_0_5 := FALSE;
    GVL_Abox.uaAboxInterface.uaDigitalOut.Output_0_6 := FALSE;
    GVL_Abox.uaAboxInterface.uaDigitalOut.Output_0_7 := FALSE;
    
    GVL_Abox.uaAboxInterface.uaDigitalOut.Output_1_0 := FALSE;
    GVL_Abox.uaAboxInterface.uaDigitalOut.Output_1_1 := FALSE;
    GVL_Abox.uaAboxInterface.uaDigitalOut.Output_1_2 := FALSE;
    GVL_Abox.uaAboxInterface.uaDigitalOut.Output_1_3 := FALSE;
    GVL_Abox.uaAboxInterface.uaDigitalOut.Output_1_4 := FALSE;
    GVL_Abox.uaAboxInterface.uaDigitalOut.Output_1_5 := FALSE;
    GVL_Abox.uaAboxInterface.uaDigitalOut.Output_1_6 := FALSE;
    GVL_Abox.uaAboxInterface.uaDigitalOut.Output_1_7 := FALSE;
    
    GVL_Abox.uaAboxInterface.uaDigitalOut.Output_2_0 := FALSE;
    GVL_Abox.uaAboxInterface.uaDigitalOut.Output_2_1 := FALSE;
    GVL_Abox.uaAboxInterface.uaDigitalOut.Output_2_2 := FALSE;
    GVL_Abox.uaAboxInterface.uaDigitalOut.Output_2_3 := FALSE;
    GVL_Abox.uaAboxInterface.uaDigitalOut.Output_2_4 := FALSE;
    GVL_Abox.uaAboxInterface.uaDigitalOut.Output_2_5 := FALSE;
    GVL_Abox.uaAboxInterface.uaDigitalOut.Output_2_6 := FALSE;
    GVL_Abox.uaAboxInterface.uaDigitalOut.Output_2_7 := FALSE;

    GVL_Abox.uaAboxInterface.uaDigitalOut.Output_3_0 := FALSE;
    GVL_Abox.uaAboxInterface.uaDigitalOut.Output_3_1 := FALSE;
    GVL_Abox.uaAboxInterface.uaDigitalOut.Output_3_2 := FALSE;
    GVL_Abox.uaAboxInterface.uaDigitalOut.Output_3_3 := FALSE;
    GVL_Abox.uaAboxInterface.uaDigitalOut.Output_3_4 := FALSE;
    GVL_Abox.uaAboxInterface.uaDigitalOut.Output_3_5 := FALSE;
    GVL_Abox.uaAboxInterface.uaDigitalOut.Output_3_6 := FALSE;
    GVL_Abox.uaAboxInterface.uaDigitalOut.Output_3_7 := FALSE;	
END_IF

IF GVL_Abox.uaAboxInterface.uaButtonAndSignal.In_Reset AND
   GVL_Abox.uaAboxInterface.uaButtonAndSignal.In_Start AND
   GVL_Abox.uaAboxInterface.uaButtonAndSignal.In_Stop  THEN
	NotResetTest := TRUE;
END_IF


IF NotResetTest THEN 
	
	// Quick Blink
	clignote(IN := changeMe,
			 PT := T#500MS);
			 
	IF clignote.Q THEN
		changeMe := FALSE;
	ELSE
		changeMe := TRUE;
	END_IF

	// Slow Blink
	clignoteSlow(IN := changeMeSlow,
			 	 PT := T#2500MS);
			 
	IF clignoteSlow.Q THEN
		changeMeSlow := FALSE;
	ELSE
		changeMeSlow := TRUE;
	END_IF
	
	IF (NOT GVL_Abox.uaAboxInterface.uaSchunkGripper.SetOut) AND clignoteSlow.Q THEN
		GVL_Abox.uaAboxInterface.uaSchunkGripper.SetOut := TRUE;
	ELSIF GVL_Abox.uaAboxInterface.uaSchunkGripper.SetOut AND clignoteSlow.Q THEN
		GVL_Abox.uaAboxInterface.uaSchunkGripper.SetOut := FALSE;
	END_IF
	
	IF (NOT GVL_Abox.uaAboxInterface.uaDigitalOut.Output_0_0) AND clignote.Q THEN
		GVL_Abox.uaAboxInterface.uaButtonAndSignal.Out_Execute := TRUE;	
		GVL_Abox.uaAboxInterface.uaButtonAndSignal.Out_Idle := TRUE;	
		GVL_Abox.uaAboxInterface.uaButtonAndSignal.Out_Stopped := TRUE;	
	
		GVL_Abox.uaAboxInterface.uaDigitalOut.Output_0_0 := TRUE;
		GVL_Abox.uaAboxInterface.uaDigitalOut.Output_0_1 := TRUE;
		GVL_Abox.uaAboxInterface.uaDigitalOut.Output_0_2 := TRUE;
		GVL_Abox.uaAboxInterface.uaDigitalOut.Output_0_3 := TRUE;
		GVL_Abox.uaAboxInterface.uaDigitalOut.Output_0_4 := TRUE;
		GVL_Abox.uaAboxInterface.uaDigitalOut.Output_0_5 := TRUE;
		GVL_Abox.uaAboxInterface.uaDigitalOut.Output_0_6 := TRUE;
		GVL_Abox.uaAboxInterface.uaDigitalOut.Output_0_7 := TRUE;
		
		GVL_Abox.uaAboxInterface.uaDigitalOut.Output_1_0 := TRUE;
		GVL_Abox.uaAboxInterface.uaDigitalOut.Output_1_1 := TRUE;
		GVL_Abox.uaAboxInterface.uaDigitalOut.Output_1_2 := TRUE;
		GVL_Abox.uaAboxInterface.uaDigitalOut.Output_1_3 := TRUE;
		GVL_Abox.uaAboxInterface.uaDigitalOut.Output_1_4 := TRUE;
		GVL_Abox.uaAboxInterface.uaDigitalOut.Output_1_5 := TRUE;
		GVL_Abox.uaAboxInterface.uaDigitalOut.Output_1_6 := TRUE;
		GVL_Abox.uaAboxInterface.uaDigitalOut.Output_1_7 := TRUE;
		
		GVL_Abox.uaAboxInterface.uaDigitalOut.Output_2_0 := TRUE;
		GVL_Abox.uaAboxInterface.uaDigitalOut.Output_2_1 := TRUE;
		GVL_Abox.uaAboxInterface.uaDigitalOut.Output_2_2 := TRUE;
		GVL_Abox.uaAboxInterface.uaDigitalOut.Output_2_3 := TRUE;
		GVL_Abox.uaAboxInterface.uaDigitalOut.Output_2_4 := TRUE;
		GVL_Abox.uaAboxInterface.uaDigitalOut.Output_2_5 := TRUE;
		GVL_Abox.uaAboxInterface.uaDigitalOut.Output_2_6 := TRUE;
		GVL_Abox.uaAboxInterface.uaDigitalOut.Output_2_7 := TRUE;

		GVL_Abox.uaAboxInterface.uaDigitalOut.Output_3_0 := TRUE;
		GVL_Abox.uaAboxInterface.uaDigitalOut.Output_3_1 := TRUE;
		GVL_Abox.uaAboxInterface.uaDigitalOut.Output_3_2 := TRUE;
		GVL_Abox.uaAboxInterface.uaDigitalOut.Output_3_3 := TRUE;
		GVL_Abox.uaAboxInterface.uaDigitalOut.Output_3_4 := TRUE;
		GVL_Abox.uaAboxInterface.uaDigitalOut.Output_3_5 := TRUE;
		GVL_Abox.uaAboxInterface.uaDigitalOut.Output_3_6 := TRUE;
		GVL_Abox.uaAboxInterface.uaDigitalOut.Output_3_7 := TRUE;
	ELSIF GVL_Abox.uaAboxInterface.uaDigitalOut.Output_0_0 AND clignote.Q THEN
		GVL_Abox.uaAboxInterface.uaButtonAndSignal.Out_Execute := FALSE;	
		GVL_Abox.uaAboxInterface.uaButtonAndSignal.Out_Idle := FALSE;	
		GVL_Abox.uaAboxInterface.uaButtonAndSignal.Out_Stopped := FALSE;	

		GVL_Abox.uaAboxInterface.uaDigitalOut.Output_0_0 := FALSE;
		GVL_Abox.uaAboxInterface.uaDigitalOut.Output_0_1 := FALSE;
		GVL_Abox.uaAboxInterface.uaDigitalOut.Output_0_2 := FALSE;
		GVL_Abox.uaAboxInterface.uaDigitalOut.Output_0_3 := FALSE;
		GVL_Abox.uaAboxInterface.uaDigitalOut.Output_0_4 := FALSE;
		GVL_Abox.uaAboxInterface.uaDigitalOut.Output_0_5 := FALSE;
		GVL_Abox.uaAboxInterface.uaDigitalOut.Output_0_6 := FALSE;
		GVL_Abox.uaAboxInterface.uaDigitalOut.Output_0_7 := FALSE;
		
		GVL_Abox.uaAboxInterface.uaDigitalOut.Output_1_0 := FALSE;
		GVL_Abox.uaAboxInterface.uaDigitalOut.Output_1_1 := FALSE;
		GVL_Abox.uaAboxInterface.uaDigitalOut.Output_1_2 := FALSE;
		GVL_Abox.uaAboxInterface.uaDigitalOut.Output_1_3 := FALSE;
		GVL_Abox.uaAboxInterface.uaDigitalOut.Output_1_4 := FALSE;
		GVL_Abox.uaAboxInterface.uaDigitalOut.Output_1_5 := FALSE;
		GVL_Abox.uaAboxInterface.uaDigitalOut.Output_1_6 := FALSE;
		GVL_Abox.uaAboxInterface.uaDigitalOut.Output_1_7 := FALSE;
		
		GVL_Abox.uaAboxInterface.uaDigitalOut.Output_2_0 := FALSE;
		GVL_Abox.uaAboxInterface.uaDigitalOut.Output_2_1 := FALSE;
		GVL_Abox.uaAboxInterface.uaDigitalOut.Output_2_2 := FALSE;
		GVL_Abox.uaAboxInterface.uaDigitalOut.Output_2_3 := FALSE;
		GVL_Abox.uaAboxInterface.uaDigitalOut.Output_2_4 := FALSE;
		GVL_Abox.uaAboxInterface.uaDigitalOut.Output_2_5 := FALSE;
		GVL_Abox.uaAboxInterface.uaDigitalOut.Output_2_6 := FALSE;
		GVL_Abox.uaAboxInterface.uaDigitalOut.Output_2_7 := FALSE;

		GVL_Abox.uaAboxInterface.uaDigitalOut.Output_3_0 := FALSE;
		GVL_Abox.uaAboxInterface.uaDigitalOut.Output_3_1 := FALSE;
		GVL_Abox.uaAboxInterface.uaDigitalOut.Output_3_2 := FALSE;
		GVL_Abox.uaAboxInterface.uaDigitalOut.Output_3_3 := FALSE;
		GVL_Abox.uaAboxInterface.uaDigitalOut.Output_3_4 := FALSE;
		GVL_Abox.uaAboxInterface.uaDigitalOut.Output_3_5 := FALSE;
		GVL_Abox.uaAboxInterface.uaDigitalOut.Output_3_6 := FALSE;
		GVL_Abox.uaAboxInterface.uaDigitalOut.Output_3_7 := FALSE;
	END_IF;
END_IF
                  
END_PROGRAM

FUNCTION_BLOCK FB_PackStates
  VAR_INPUT
    Enable : BOOL;
    SoftEstop : BOOL;
    Hold : BOOL := FALSE;
    Unhold : BOOL := FALSE;
    Clearing_SC : BOOL := TRUE;
    Stopping_SC : BOOL := TRUE;
    Aborting_SC : BOOL := TRUE;
    Resetting_SC : BOOL := TRUE;
    Starting_SC : BOOL := TRUE;
    Execute_SC : BOOL := FALSE;
    Holding_SC : BOOL := FALSE;
    Unholding_SC : BOOL := FALSE;
  END_VAR
  VAR_IN_OUT
    remote : UA_ButtonAndSignal;
  END_VAR
  VAR_OUTPUT
    state : ST_PackState;
    strState : STRING;
  END_VAR
  VAR
    initialized : BOOL;
    ePackStates : E_PackStates;
    rTrigStop : R_TRIG;
    rTrigStart : R_TRIG;
    rTrigReset : R_TRIG;
    clignote : TON;
    changeMe : BOOL;
  END_VAR

                    // 
//	Init
//
IF Enable THEN
	IF NOT initialized THEN
		// Init at Aborted when entering state machine.
		initialized := TRUE;
		ePackStates := E_PackStates.Aborted;
	END_IF;
ELSE
	ePackStates := E_PackStates.NotActive;
	initialized := FALSE;
END_IF

//
//	Manage Inputs
//
rTrigStop(CLK := remote.In_Stop);
rTrigStart(CLK := remote.In_Start);
rTrigReset(CLK := remote.In_Reset);

CASE ePackStates OF
	E_PackStates.NotActive	:
		strState := 'Not Active';
		;
	E_PackStates.Aborting 	:;
		strState := 'Aborting';
		IF Aborting_SC THEN
			ePackStates := E_PackStates.Aborted;
		END_IF
		
	E_PackStates.Aborted 	:
		strState := 'Aborted';
		IF rTrigReset.Q THEN
			ePackStates := E_PackStates.Clearing;
		END_IF
	
	E_PackStates.Clearing 	:
		strState := 'Clearing';
		// E-Stop Active Low
		IF NOT remote.In_Estop OR SoftEstop THEN
			ePackStates := E_PackStates.Aborting;
		ELSIF Clearing_SC THEN
			ePackStates := E_PackStates.Stopped;	
		END_IF

	E_PackStates.Stopped 	:
		strState := 'Stopped';
		// E-Stop Active Low
		IF NOT remote.In_Estop OR SoftEstop THEN
			ePackStates := E_PackStates.Aborting;
		ELSIF rTrigReset.Q THEN
			ePackStates := E_PackStates.Resetting;
		END_IF

	E_PackStates.Stopping 	:
		strState := 'Stopping';
		// E-Stop Active Low
		IF NOT remote.In_Estop OR SoftEstop THEN
			ePackStates := E_PackStates.Aborting;
		ELSIF Stopping_SC THEN
			ePackStates := E_PackStates.Stopped;
		END_IF

	E_PackStates.Resetting 	:
		strState := 'Resetting';
		// E-Stop Active Low
		IF NOT remote.In_Estop OR SoftEstop THEN
			ePackStates := E_PackStates.Aborting;
		ELSIF rTrigStop.Q THEN
			ePackStates := E_PackStates.Stopping;
		ELSIF Resetting_SC THEN
			ePackStates := E_PackStates.Idle;			
		END_IF

	E_PackStates.Idle 		:
		strState := 'Idle';
		// E-Stop Active Low
		IF NOT remote.In_Estop OR SoftEstop THEN
			ePackStates := E_PackStates.Aborting;
		ELSIF rTrigStop.Q THEN
			ePackStates := E_PackStates.Stopping;
		ELSIF rTrigStart.Q THEN
			ePackStates := E_PackStates.Starting;
		END_IF

	E_PackStates.Starting 	:
		strState := 'Starting';
		// E-Stop Active Low
		IF NOT remote.In_Estop OR SoftEstop THEN
			ePackStates := E_PackStates.Aborting;
		ELSIF rTrigStop.Q THEN
			ePackStates := E_PackStates.Stopping;
		ELSIF Starting_SC THEN
			ePackStates := E_PackStates.Execute;	
		END_IF

	E_PackStates.Execute 	:
		strState := 'Execute';
		// E-Stop Active Low
		IF NOT remote.In_Estop OR SoftEstop THEN
			ePackStates := E_PackStates.Aborting;
		ELSIF rTrigStop.Q THEN
			ePackStates := E_PackStates.Stopping;
		ELSIF Hold		 THEN
			ePackStates := E_PackStates.Holding;	
		ELSIF Execute_SC THEN
			ePackStates := E_PackStates.Execute;	
		END_IF
		
	(* Held Loop *)
	E_PackStates.Holding	:;
		strState := 'Holding';
		// E-Stop Active Low
		IF NOT remote.In_Estop OR SoftEstop THEN
			ePackStates := E_PackStates.Aborting;
		ELSIF rTrigStop.Q THEN
			ePackStates := E_PackStates.Stopping;
		ELSIF Holding_SC THEN
			ePackStates := E_PackStates.Held;	
		END_IF
		
	E_PackStates.Held		:;
		strState := 'Held';
		// E-Stop Active Low
		IF NOT remote.In_Estop OR SoftEstop THEN
			ePackStates := E_PackStates.Aborting;
		ELSIF rTrigStop.Q THEN
			ePackStates := E_PackStates.Stopping;
		ELSIF Unhold THEN
			ePackStates := E_PackStates.Unholding;	
		END_IF

	E_PackStates.Unholding	:;
		strState := 'Unholding';
		// E-Stop Active Low
		IF NOT remote.In_Estop OR SoftEstop THEN
			ePackStates := E_PackStates.Aborting;
		ELSIF rTrigStop.Q THEN
			ePackStates := E_PackStates.Stopping;
		ELSIF Unholding_SC THEN
			ePackStates := E_PackStates.Execute;	
		END_IF

END_CASE

// Quick Blink
clignote(IN := changeMe,
		 PT := T#500MS);
			 
IF clignote.Q THEN
	changeMe := FALSE;
ELSE
	changeMe := TRUE;
END_IF

// Set Output states
state.Aborting	:= (ePackStates = E_PackStates.Aborting);
state.Aborted	:= (ePackStates = E_PackStates.Aborted);
state.Clearing	:= (ePackStates = E_PackStates.Clearing);
state.Stopped	:= (ePackStates = E_PackStates.Stopped);
state.Stopping	:= (ePackStates = E_PackStates.Stopping);
state.Resetting	:= (ePackStates = E_PackStates.Resetting);
state.Idle		:= (ePackStates = E_PackStates.Idle);
state.Starting	:= (ePackStates = E_PackStates.Starting);
state.Execute	:= (ePackStates = E_PackStates.Execute);

// Set Output signals
remote.Out_Stopped := (ePackStates = E_PackStates.Stopped);

IF ePackStates = E_PackStates.Starting THEN
	IF remote.Out_Execute AND clignote.Q THEN
		remote.Out_Execute := FALSE;
	ELSIF NOT remote.Out_Execute AND clignote.Q THEN
		remote.Out_Execute := TRUE;
	END_IF
ELSE
	remote.Out_Execute := (ePackStates = E_PackStates.Execute);	
END_IF

IF ePackStates = E_PackStates.Resetting THEN
	IF remote.Out_Idle AND clignote.Q THEN
		remote.Out_Idle := FALSE;
	ELSIF NOT remote.Out_Idle AND clignote.Q THEN
		remote.Out_Idle := TRUE;
	END_IF
ELSE
	remote.Out_Idle := (ePackStates = E_PackStates.Idle);	
END_IF

IF ePackStates = E_PackStates.Stopping OR 
   ePackStates = E_PackStates.Clearing THEN
	IF remote.Out_Stopped AND clignote.Q THEN
		remote.Out_Stopped := FALSE;
	ELSIF NOT remote.Out_Stopped AND clignote.Q THEN
		remote.Out_Stopped := TRUE;
	END_IF
ELSE
	remote.Out_Stopped := (ePackStates = E_PackStates.Stopped);	
END_IF
                  
END_FUNCTION_BLOCK

FUNCTION_BLOCK FB_GenerateProfile
  VAR_INPUT
    bStartForward : BOOL;  (* Start of motion at rising edge. *)
    bStartBackward : BOOL;
    startPosition_mm : LREAL := 0;  (* Should be 0 for first version, could be extended for any position *)
    endPosition_mm : LREAL := 0;  (* Should be limited to 100 mm *)
    udiCyclTime_ms : UDINT;  (* Cycle time in ms of the task where FB is running. *)
    udiCycleTimeMult : UDINT;  (* Cycle time multiplier, used to compute duration of motion This could be made automatically later, Now result in Output *)
  END_VAR
  VAR_IN_OUT
    arGoToPos : ARRAY[0..GVL_CyclSetPoint.c_uiMaxProfilePoints] OF LREAL;  (* Used for verification of data, we do not nead them for motion *)
    arReturnFromPos : ARRAY[0..GVL_CyclSetPoint.c_uiMaxProfilePoints] OF LREAL;  (* Used for verification of data, we do not nead them for motion *)
  END_VAR
  VAR_OUTPUT
    udiMotionTime_ms : UDINT;  (* Is time to execute the profile in ms Multiplication of udiCyclTime_ms x udiCycleTimeMult *)
    bDoneForward : BOOL;  (* Motion finished *)
    bDoneBackward : BOOL;
    lrSetPosition : LREAL;  (* Motion set position *)
    bErrorTimeMultToBig : BOOL;  (* True if udiCycleTimeMult Exceeds, FB not executed *)
    bActive : BOOL;  (* Point generator active *)
  END_VAR
  VAR
    discreteTimeIndex : UDINT;  (* Time index of position *)
    rStartForward : R_TRIG;  (* rising edge of start *)
    rStartBackward : R_TRIG;
    lrTimeScaler : LREAL;  (* Ce machin là va devoir être expliqué avec pas mal de détail en théorie. *)
  END_VAR

                    rStartForward(clk := bStartForward);
rStartBackward(clk := bStartBackward);


udiMotionTime_ms := udiCyclTime_ms * udiCycleTimeMult;

IF udiCycleTimeMult > GVL_CyclSetPoint.c_uiMaxProfilePoints THEN
    bErrorTimeMultToBig := TRUE;
    bActive := FALSE;
    bDoneForward := FALSE;
    bDoneBackward := FALSE;
ELSE
    IF bStartForward THEN
        // Init motion
        IF rStartForward.Q THEN
            lrSetPosition := startPosition_mm;
            discreteTimeIndex := 0; 
            lrTimeScaler := 1/UDINT_TO_LREAL(udiCycleTimeMult);
            bActive := TRUE;
            bDoneForward := FALSE;
        END_IF // rStartForward.Q
        
        IF NOT bDoneForward THEN
            // Matlab operation with some modifications : 
            // position_yAxis(iLoop) = (t_xAxis(iLoop)^3 * P5_position(4) + t_xAxis(iLoop)^4 * P5_position(5) + t_xAxis(iLoop)^5 * P5_position(6)) * y_scaling_mm;
            arGoToPos[discreteTimeIndex] := startPosition_mm                                                 + 
											(EXPT(lrTimeScaler*discreteTimeIndex,3) * GVL_CyclSetPoint.P5[4] +
                                             EXPT(lrTimeScaler*discreteTimeIndex,4) * GVL_CyclSetPoint.P5[5] +
                                             EXPT(lrTimeScaler*discreteTimeIndex,5) * GVL_CyclSetPoint.P5[6]) * (endPosition_mm - startPosition_mm);
            // Set new value
            lrSetPosition := arGoToPos[discreteTimeIndex];
            // inc at each cycle
            discreteTimeIndex := discreteTimeIndex + 1;
            IF discreteTimeIndex > udiCycleTimeMult THEN
                bDoneForward := TRUE;
            END_IF // discreteTimeIndex > udiCycleTimeMult
        END_IF // IF bDoneForward 
	ELSE
		bDoneForward := FALSE;		
    END_IF    

    IF bStartBackward THEN
        // Init motion
        IF rStartBackward.Q THEN
            lrSetPosition := startPosition_mm;
            discreteTimeIndex := 0; 
            lrTimeScaler := 1/UDINT_TO_LREAL(udiCycleTimeMult);
            bActive := TRUE;
            bDoneBackward := FALSE;
        END_IF // rStartForward.Q
        
        IF NOT bDoneBackward THEN
            // Matlab operation with some modifications : 
            // position_yAxisBack(iLoop) = y_scaling_mm - (t_xAxis(iLoop)^3 * P5_position(4) + t_xAxis(iLoop)^4 * P5_position(5) + t_xAxis(iLoop)^5 * P5_position(6)) * y_scaling_mm;
            arReturnFromPos[discreteTimeIndex] := endPosition_mm - (EXPT(lrTimeScaler*discreteTimeIndex,3) * GVL_CyclSetPoint.P5[4] +
                                                                    EXPT(lrTimeScaler*discreteTimeIndex,4) * GVL_CyclSetPoint.P5[5] +
                                                                    EXPT(lrTimeScaler*discreteTimeIndex,5) * GVL_CyclSetPoint.P5[6]) * (endPosition_mm - startPosition_mm);
            // Set new value
            lrSetPosition := arReturnFromPos[discreteTimeIndex];
            // inc at each cycle
            discreteTimeIndex := discreteTimeIndex + 1;
            IF discreteTimeIndex > udiCycleTimeMult THEN
                bDoneBackward := TRUE;
            END_IF // discreteTimeIndex > udiCycleTimeMult
        END_IF // IF bDoneBackward 
	ELSE
		bDoneBackward := FALSE;		
    END_IF    

END_IF

                  
END_FUNCTION_BLOCK

CONFIGURATION PracticalWork_01
  RESOURCE BaseInterfaceUa ON PLC
    {attribute 'qualified_only'}
    VAR_GLOBAL  (* GVL_Abox *)
      uaAboxInterface : UA_AboxInterface;
    END_VAR
    {attribute 'qualified_only'}
    VAR_GLOBAL  (* GVL_AxisDefines *)
      X_Axis : MB_AXISIF_REF := (AxisName := 'Axis_1', AxisNo := 1);
      Y_Axis : MB_AXISIF_REF := (AxisName := 'Axis_2', AxisNo := 2);
      Z_Axis : MB_AXISIF_REF := (AxisName := 'Axis_3', AxisNo := 3);
    END_VAR
    {attribute 'qualified_only'}
    VAR_GLOBAL  (* GVL_CyclSetPoint *)
      stRemote : ST_RemoteCyclicSetPosition := (in := (lrStartPosition_mm := 50, lrEndPosition_mm := 100));  (* Remote for this program *)
      arGoToPosition : ARRAY[0..c_uiMaxProfilePoints] OF LREAL;  (* These values are for check only, it is possible to work without buffer *)
      arReturnFromPosition : ARRAY[0..c_uiMaxProfilePoints] OF LREAL;
      c_uiMaxProfilePoints : UDINT := 1000;  (* 1001 points of 2 ms for max 2 [s] motion *)
      P5 : ARRAY[1..6] OF LREAL := [0, 0, 0, 10, -15, 6];  (* P5 Polynomial P5(0) to P5(5) exp 0 to 5 *)
      MOTION_CYCLE_TIME_ms : UDINT := 2;  (* equal to real time bus *)
    END_VAR
    TASK MainTask(PRIORITY := 30);
    PROGRAM PRG_CyclicSetPoint WITH MainTask : PRG_CyclicSetPoint;
    PROGRAM PRG_MapBox WITH MainTask : PRG_MapBox;
  END_RESOURCE
END_CONFIGURATION

CONFIGURATION Realtime_Data
END_CONFIGURATION
